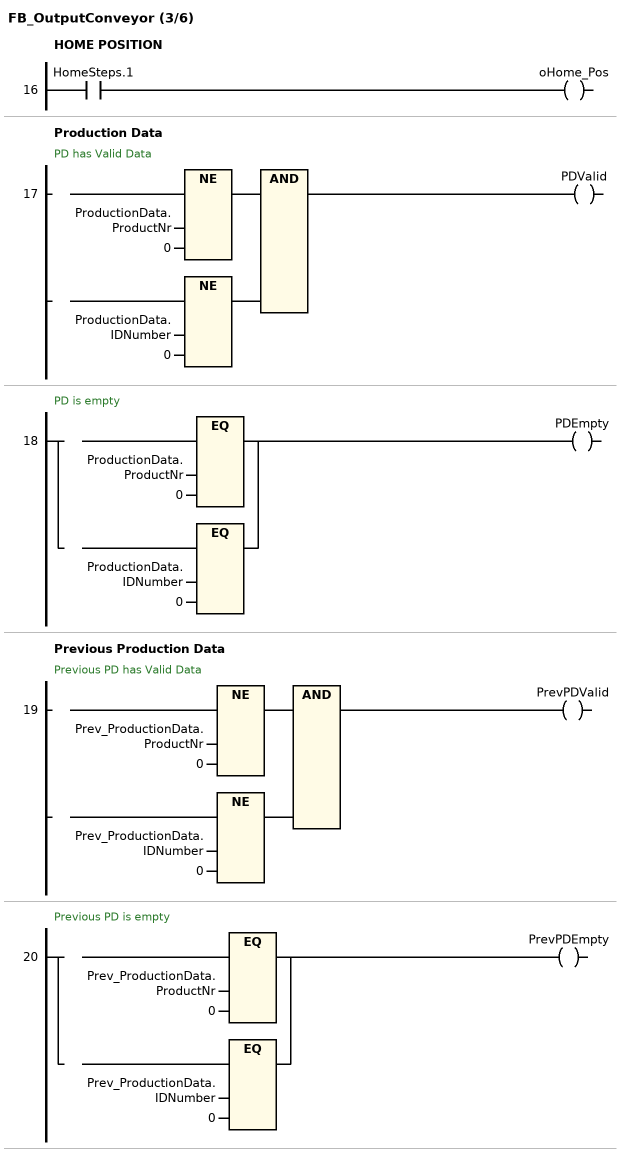
// NETWORK 16: HOME POSITION
oHome_Pos := HomeSteps.1;

// NETWORK 17: Production Data
// PD has Valid Data
PDValid := ProductionData.ProductNr <> 0 AND ProductionData.IDNumber <> 0;

// NETWORK 18
// PD is empty
PDEmpty := ProductionData.ProductNr = 0 OR ProductionData.IDNumber = 0;

// NETWORK 19: Previous Production Data
// Previous PD has Valid Data
PrevPDValid := Prev_ProductionData.ProductNr <> 0 AND Prev_ProductionData.IDNumber <> 0;

// NETWORK 20
// Previous PD is empty
PrevPDEmpty := Prev_ProductionData.ProductNr = 0 OR Prev_ProductionData.IDNumber = 0;

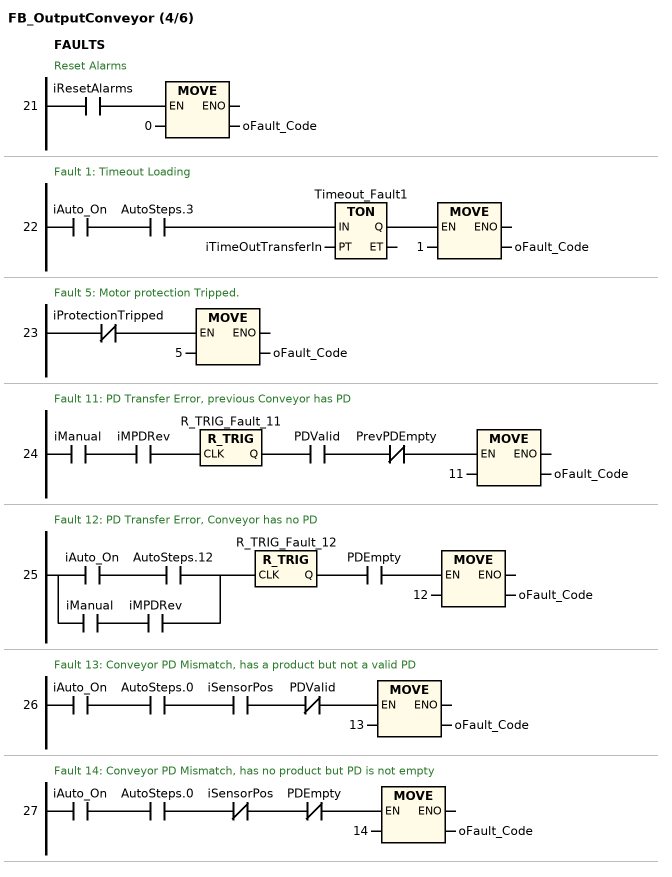
// NETWORK 21: FAULTS
// Reset Alarms
IF iResetAlarms THEN oFault_Code := 0; END_IF

// NETWORK 22
// Fault 1: Timeout Loading
Timeout_Fault1(IN := iAuto_On AND AutoSteps.3, PT := iTimeOutTransferIn); // TON
IF Timeout_Fault1.Q THEN oFault_Code := 1; END_IF

// NETWORK 23
// Fault 5: Motor protection Tripped.
IF NOT iProtectionTripped THEN oFault_Code := 5; END_IF

// NETWORK 24
// Fault 11: PD Transfer Error, previous Conveyor has PD
R_TRIG_Fault_11(CLK := iManual AND iMPDRev); // R_TRIG
IF R_TRIG_Fault_11.Q AND PDValid AND NOT PrevPDEmpty THEN oFault_Code := 11; END_IF

// NETWORK 25
// Fault 12: PD Transfer Error, Conveyor has no PD
R_TRIG_Fault_12(CLK := iAuto_On AND AutoSteps.12 OR iManual AND iMPDRev); // R_TRIG
IF R_TRIG_Fault_12.Q AND PDEmpty THEN oFault_Code := 12; END_IF

// NETWORK 26
// Fault 13: Conveyor PD Mismatch, has a product but not a valid PD
IF iAuto_On AND AutoSteps.0 AND iSensorPos AND NOT PDValid THEN oFault_Code := 13; END_IF

// NETWORK 27
// Fault 14: Conveyor PD Mismatch, has no product but PD is not empty
IF iAuto_On AND AutoSteps.0 AND NOT iSensorPos AND NOT PDEmpty THEN oFault_Code := 14; END_IF

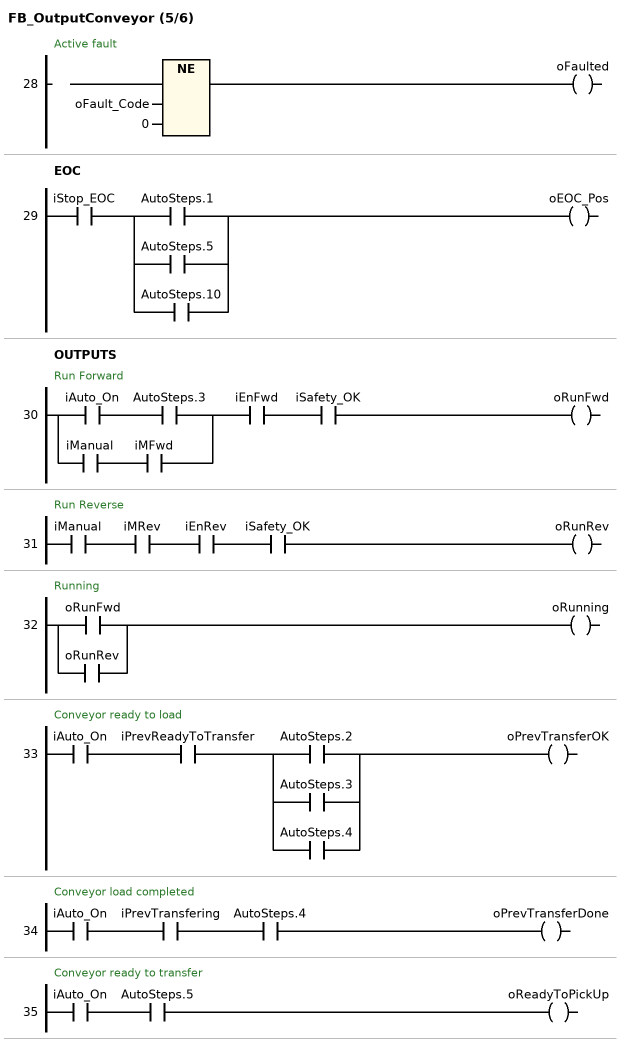
// NETWORK 28
// Active fault
oFaulted := oFault_Code <> 0;

// NETWORK 29: EOC
oEOC_Pos := iStop_EOC AND (AutoSteps.1 OR AutoSteps.5 OR AutoSteps.10);

// NETWORK 30: OUTPUTS
// Run Forward
oRunFwd := (iAuto_On AND AutoSteps.3 OR iManual AND iMFwd) AND iEnFwd AND iSafety_OK;

// NETWORK 31
// Run Reverse
oRunRev := iManual AND iMRev AND iEnRev AND iSafety_OK;

// NETWORK 32
// Running
oRunning := oRunFwd OR oRunRev;

// NETWORK 33
// Conveyor ready to load
oPrevTransferOK := iAuto_On AND iPrevReadyToTransfer AND (AutoSteps.2 OR AutoSteps.3 OR AutoSteps.4);

// NETWORK 34
// Conveyor load completed
oPrevTransferDone := iAuto_On AND iPrevTransfering AND AutoSteps.4;

// NETWORK 35
// Conveyor ready to transfer
oReadyToPickUp := iAuto_On AND AutoSteps.5;

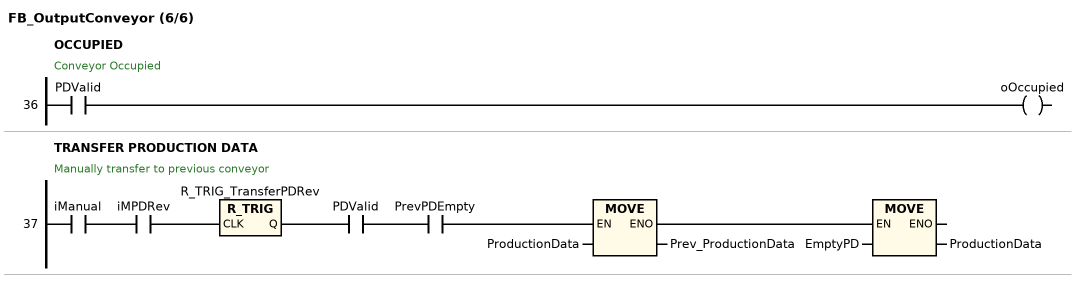
// NETWORK 36: OCCUPIED
// Conveyor Occupied
oOccupied := PDValid;

// NETWORK 37: TRANSFER PRODUCTION DATA
// Manually transfer to previous conveyor
R_TRIG_TransferPDRev(CLK := iManual AND iMPDRev); // R_TRIG
_w13 := R_TRIG_TransferPDRev.Q AND PDValid AND PrevPDEmpty;
IF _w13 THEN Prev_ProductionData := ProductionData; END_IF
IF _w13 THEN ProductionData := EmptyPD; END_IF

END_FUNCTION_BLOCK

// Device/Application/SOP670
PROGRAM SOP670
VAR
END_VAR

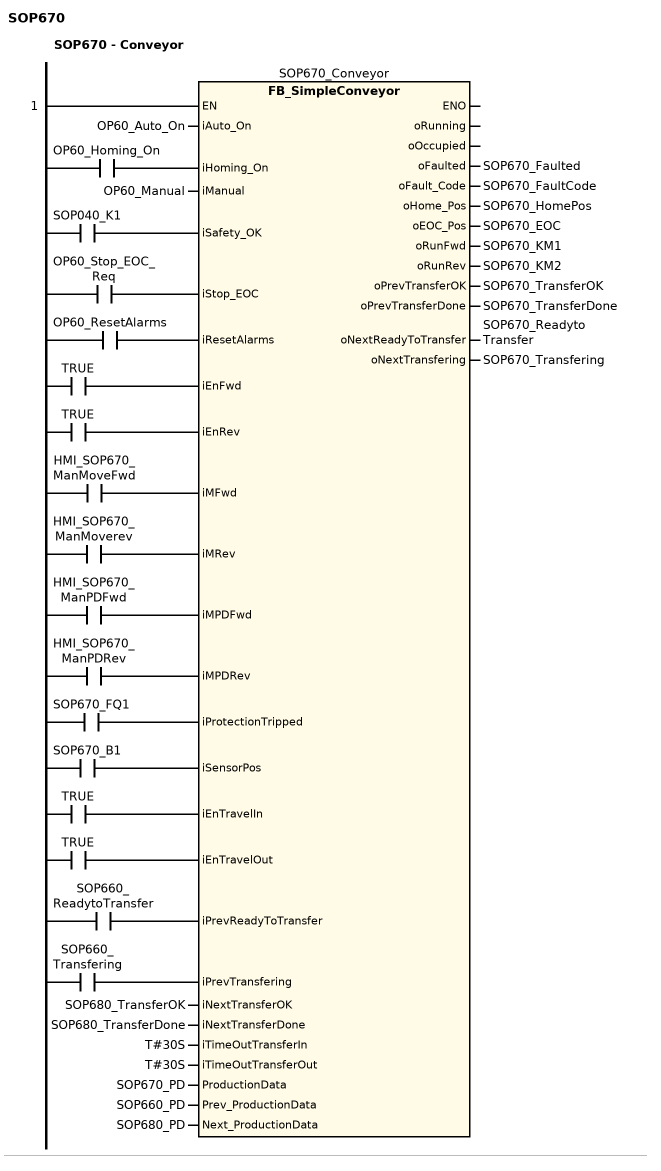
// NETWORK 1: SOP670 - Conveyor
SOP670_Conveyor(
    iAuto_On := OP60_Auto_On,
    iHoming_On := OP60_Homing_On,
    iManual := OP60_Manual,
    iSafety_OK := SOP040_K1,
    iStop_EOC := OP60_Stop_EOC_Req,
    iResetAlarms := OP60_ResetAlarms,
    iEnFwd := TRUE,
    iEnRev := TRUE,
    iMFwd := HMI_SOP670_ManMoveFwd,
    iMRev := HMI_SOP670_ManMoverev,
    iMPDFwd := HMI_SOP670_ManPDFwd,
    iMPDRev := HMI_SOP670_ManPDRev,
    iProtectionTripped := SOP670_FQ1,
    iSensorPos := SOP670_B1,
    iEnTravelIn := TRUE,
    iEnTravelOut := TRUE,
    iPrevReadyToTransfer := SOP660_ReadytoTransfer,
    iPrevTransfering := SOP660_Transfering,
    iNextTransferOK := SOP680_TransferOK,
    iNextTransferDone := SOP680_TransferDone,
    iTimeOutTransferIn := T#30S,
    iTimeOutTransferOut := T#30S,
    ProductionData := SOP670_PD,
    Prev_ProductionData := SOP660_PD,
    Next_ProductionData := SOP680_PD,
    oFaulted => SOP670_Faulted,
    oFault_Code => SOP670_FaultCode,
    oHome_Pos => SOP670_HomePos,
    oEOC_Pos => SOP670_EOC,
    oRunFwd => SOP670_KM1,
    oRunRev => SOP670_KM2,
    oPrevTransferOK => SOP670_TransferOK,
    oPrevTransferDone => SOP670_TransferDone,
    oNextReadyToTransfer => SOP670_ReadytoTransfer,
    oNextTransfering => SOP670_Transfering); // FB_SimpleConveyor

END_PROGRAM

// Device/Application/FBs/FB_SimpleConveyor
FUNCTION_BLOCK FB_SimpleConveyor
VAR_INPUT
	iAuto_On: BOOL; // Auto-On cycle active
	iHoming_On: BOOL; // Homing-On cycle active
	iManual: BOOL; // Manual mode active
	iSafety_OK: BOOL; // Safety circuit OK
	iStop_EOC: BOOL; // Stop EOC selected
	iResetAlarms: BOOL; // Reset Alarms
	
	iEnFwd: BOOL := TRUE; // Interlock signal movement forward
	iEnRev: BOOL := TRUE; // Interlock signal movement reverse
	
	iMFwd: BOOL; 	// Manual Fwd request
	iMRev: BOOL; 	// Manual Rev request
	iMPDFwd: BOOL; 	// Manual Move PD forward
	iMPDRev: BOOL; 	// Manual Move PD reverse
	
	iProtectionTripped: BOOL := FALSE; // Motor Protection Tripped
	
	iSensorPos: BOOL; // Product in position
	
	iEnTravelIn: BOOL := TRUE; // Enable product transfer from previous conveyor.
	iEnTravelOut: BOOL := TRUE; // Enable product transfer to next conveyor.
	
	iPrevReadyToTransfer: BOOL; // Previous conveyor ready to transfer
	iPrevTransfering: BOOL; // Previous conveyor transfering
	iNextTransferOK: BOOL; // Next conveyor ready to load
	iNextTransferDone: BOOL;  // Next conveyor transfer done
	
	iTimeOutTransferIn: TIME := T#10S; // Time out time for transfer in
	iTimeOutTransferOut: TIME := T#10S; // Time out time for transfer out
END_VAR
VAR_IN_OUT
	ProductionData: ProductionData; 		// Production Data
	Prev_ProductionData: ProductionData;	// Previous Production Data
	Next_ProductionData: ProductionData;	// Next Production Data
END_VAR
VAR_OUTPUT
	oRunning: BOOL; // Conveyor Running
	oOccupied: BOOL; // Conveyor Occupied
	oFaulted : BOOL; // Conveyor faulted
	oFault_Code: INT; // Conveyor fault code
	oHome_Pos: BOOL; // Conveyor Home Position reached
	oEOC_Pos: BOOL; // Conveyor Stop EOC reached

	oRunFwd: BOOL; // Conveyor running forward
	oRunRev: BOOL; // Conveyor running reverse	

	oPrevTransferOK: BOOL; // Conveyor ready to load
	oPrevTransferDone: BOOL; // Conveyor load completed
	oNextReadyToTransfer: BOOL; // Conveyor ready to transfer
	oNextTransfering: BOOL; // Conveyor transfering
END_VAR
VAR
	AutoSteps: WORD;
	HomeSteps: WORD;
	
	Timeout_Fault1: TON;
	Timeout_Fault2: TON;
	
	EmptyPD: ProductionData;
	PDValid: BOOL;		// PD is Valid
	PDEmpty: BOOL;		// PD is Empty
	PrevPDValid: BOOL;	// Previous PD is Valid
	PrevPDEmpty: BOOL;	// Previous PD is Empty
	NextPDValid: BOOL;	// Next PD is Valid
	NextPDEmpty: BOOL;	// Next PD is Empty
	R_TRIG_TransferPDFwd: R_TRIG;
	R_TRIG_TransferPDRev: R_TRIG;
	R_TRIG_Fault_10: R_TRIG;
	R_TRIG_Fault_11: R_TRIG;
	R_TRIG_Fault_12: R_TRIG;
END_VAR
VAR // added by the converter: edge detectors and wires of the graphical bodies
    _w1, _w2, _w3, _w4, _w5, _w6, _w7, _w8, _w9, _w10, _w11, _w12, _w13, _w14, _w15, _w16 : BOOL;
END_VAR

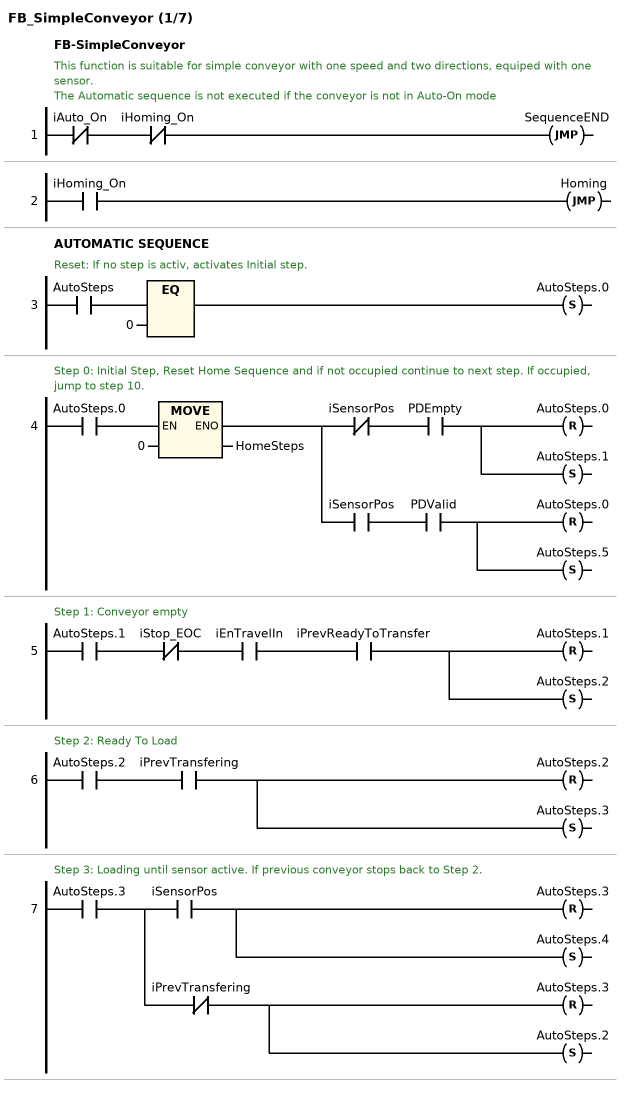
// NETWORK 1: FB-SimpleConveyor
// This function is suitable for simple conveyor with one speed and two directions, equiped with one sensor.
//
// The Automatic sequence is not executed if the conveyor is not in Auto-On mode
IF NOT iAuto_On AND NOT iHoming_On THEN JMP SequenceEND; END_IF

// NETWORK 2
IF iHoming_On THEN JMP Homing; END_IF

// NETWORK 3: AUTOMATIC SEQUENCE
// Reset: If no step is activ, activates Initial step.
AutoSteps.0 S= AutoSteps = 0;

// NETWORK 4
// Step 0: Initial Step, Reset Home Sequence and if not occupied continue to next step. If occupied, jump to step 10.
_w1 := AutoSteps.0;
IF _w1 THEN HomeSteps := 0; END_IF
_w2 := _w1 AND NOT iSensorPos AND PDEmpty;
AutoSteps.0 R= _w2;
AutoSteps.1 S= _w2;
_w3 := _w1 AND iSensorPos AND PDValid;
AutoSteps.0 R= _w3;
AutoSteps.5 S= _w3;

// NETWORK 5
// Step 1: Conveyor empty
_w4 := AutoSteps.1 AND NOT iStop_EOC AND iEnTravelIn AND iPrevReadyToTransfer;
AutoSteps.1 R= _w4;
AutoSteps.2 S= _w4;

// NETWORK 6
// Step 2: Ready To Load
_w5 := AutoSteps.2 AND iPrevTransfering;
AutoSteps.2 R= _w5;
AutoSteps.3 S= _w5;

// NETWORK 7
// Step 3: Loading until sensor active. If previous conveyor stops back to Step 2.
_w6 := AutoSteps.3;
_w7 := _w6 AND iSensorPos;
AutoSteps.3 R= _w7;
AutoSteps.4 S= _w7;
_w8 := _w6 AND NOT iPrevTransfering;
AutoSteps.3 R= _w8;
AutoSteps.2 S= _w8;

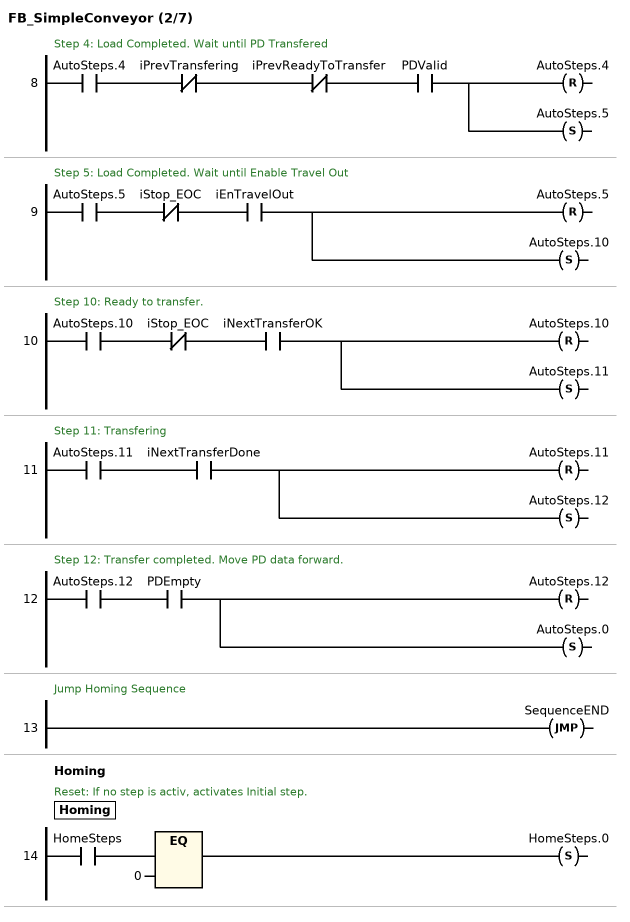
// NETWORK 8
// Step 4: Load Completed. Wait until PD Transfered
_w9 := AutoSteps.4 AND NOT iPrevTransfering AND NOT iPrevReadyToTransfer AND PDValid;
AutoSteps.4 R= _w9;
AutoSteps.5 S= _w9;

// NETWORK 9
// Step 5: Load Completed. Wait until Enable Travel Out
_w10 := AutoSteps.5 AND NOT iStop_EOC AND iEnTravelOut;
AutoSteps.5 R= _w10;
AutoSteps.10 S= _w10;

// NETWORK 10
// Step 10: Ready to transfer.
_w11 := AutoSteps.10 AND NOT iStop_EOC AND iNextTransferOK;
AutoSteps.10 R= _w11;
AutoSteps.11 S= _w11;

// NETWORK 11
// Step 11: Transfering
_w12 := AutoSteps.11 AND iNextTransferDone;
AutoSteps.11 R= _w12;
AutoSteps.12 S= _w12;

// NETWORK 12
// Step 12: Transfer completed. Move PD data forward.
_w13 := AutoSteps.12 AND PDEmpty;
AutoSteps.12 R= _w13;
AutoSteps.0 S= _w13;

// NETWORK 13
// Jump Homing Sequence
JMP SequenceEND;

// NETWORK 14: Homing
// Reset: If no step is activ, activates Initial step.
Homing:
HomeSteps.0 S= HomeSteps = 0;

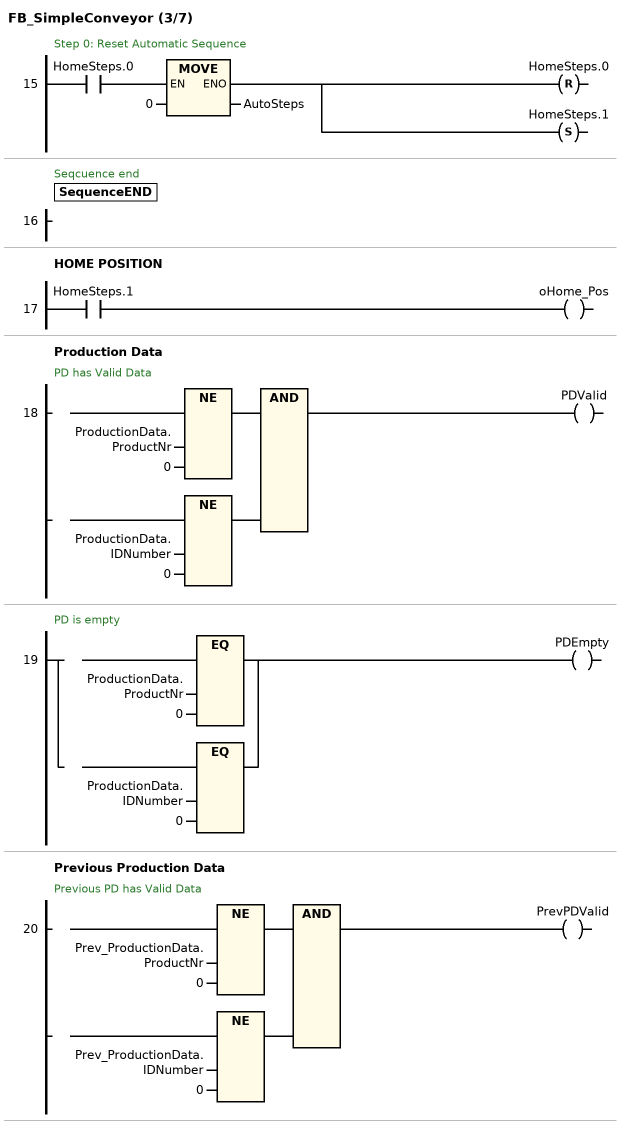
// NETWORK 15
// Step 0: Reset Automatic Sequence
_w14 := HomeSteps.0;
IF _w14 THEN AutoSteps := 0; END_IF
HomeSteps.0 R= _w14;
HomeSteps.1 S= _w14;

// NETWORK 16
// Seqcuence end
SequenceEND: ;

// NETWORK 17: HOME POSITION
oHome_Pos := HomeSteps.1;

// NETWORK 18: Production Data
// PD has Valid Data
PDValid := ProductionData.ProductNr <> 0 AND ProductionData.IDNumber <> 0;

// NETWORK 19
// PD is empty
PDEmpty := ProductionData.ProductNr = 0 OR ProductionData.IDNumber = 0;

// NETWORK 20: Previous Production Data
// Previous PD has Valid Data
PrevPDValid := Prev_ProductionData.ProductNr <> 0 AND Prev_ProductionData.IDNumber <> 0;

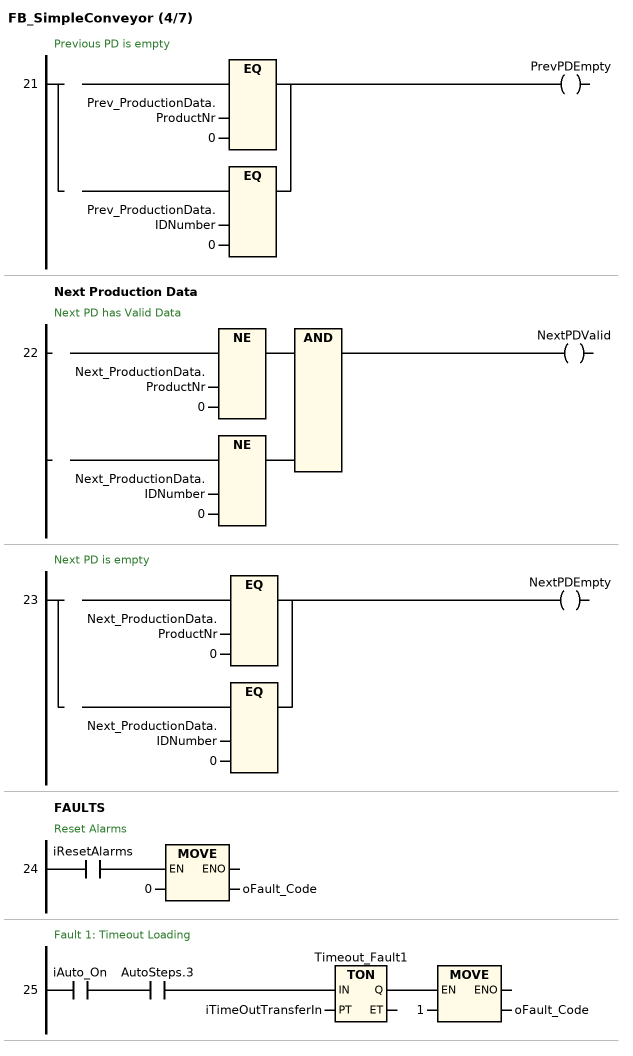
// NETWORK 21
// Previous PD is empty
PrevPDEmpty := Prev_ProductionData.ProductNr = 0 OR Prev_ProductionData.IDNumber = 0;

// NETWORK 22: Next Production Data
// Next PD has Valid Data
NextPDValid := Next_ProductionData.ProductNr <> 0 AND Next_ProductionData.IDNumber <> 0;

// NETWORK 23
// Next PD is empty
NextPDEmpty := Next_ProductionData.ProductNr = 0 OR Next_ProductionData.IDNumber = 0;

// NETWORK 24: FAULTS
// Reset Alarms
IF iResetAlarms THEN oFault_Code := 0; END_IF

// NETWORK 25
// Fault 1: Timeout Loading
Timeout_Fault1(IN := iAuto_On AND AutoSteps.3, PT := iTimeOutTransferIn); // TON
IF Timeout_Fault1.Q THEN oFault_Code := 1; END_IF

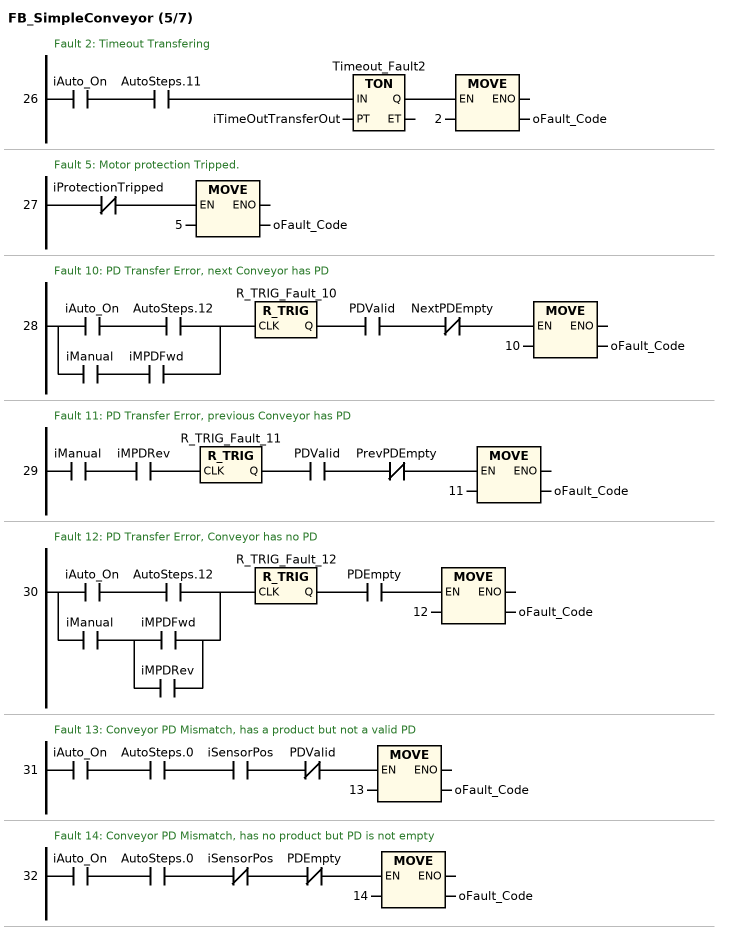
// NETWORK 26
// Fault 2: Timeout Transfering
Timeout_Fault2(IN := iAuto_On AND AutoSteps.11, PT := iTimeOutTransferOut); // TON
IF Timeout_Fault2.Q THEN oFault_Code := 2; END_IF

// NETWORK 27
// Fault 5: Motor protection Tripped.
IF NOT iProtectionTripped THEN oFault_Code := 5; END_IF

// NETWORK 28
// Fault 10: PD Transfer Error, next Conveyor has PD
R_TRIG_Fault_10(CLK := iAuto_On AND AutoSteps.12 OR iManual AND iMPDFwd); // R_TRIG
IF R_TRIG_Fault_10.Q AND PDValid AND NOT NextPDEmpty THEN oFault_Code := 10; END_IF

// NETWORK 29
// Fault 11: PD Transfer Error, previous Conveyor has PD
R_TRIG_Fault_11(CLK := iManual AND iMPDRev); // R_TRIG
IF R_TRIG_Fault_11.Q AND PDValid AND NOT PrevPDEmpty THEN oFault_Code := 11; END_IF

// NETWORK 30
// Fault 12: PD Transfer Error, Conveyor has no PD
R_TRIG_Fault_12(CLK := iAuto_On AND AutoSteps.12 OR iManual AND (iMPDFwd OR iMPDRev)); // R_TRIG
IF R_TRIG_Fault_12.Q AND PDEmpty THEN oFault_Code := 12; END_IF

// NETWORK 31
// Fault 13: Conveyor PD Mismatch, has a product but not a valid PD
IF iAuto_On AND AutoSteps.0 AND iSensorPos AND NOT PDValid THEN oFault_Code := 13; END_IF

// NETWORK 32
// Fault 14: Conveyor PD Mismatch, has no product but PD is not empty
IF iAuto_On AND AutoSteps.0 AND NOT iSensorPos AND NOT PDEmpty THEN oFault_Code := 14; END_IF

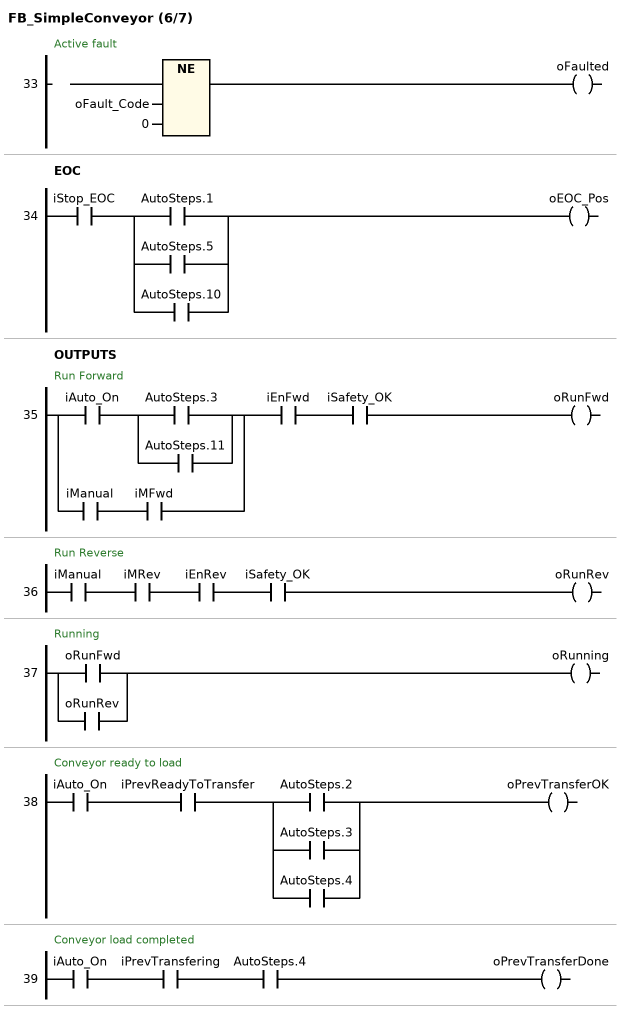
// NETWORK 33
// Active fault
oFaulted := oFault_Code <> 0;

// NETWORK 34: EOC
oEOC_Pos := iStop_EOC AND (AutoSteps.1 OR AutoSteps.5 OR AutoSteps.10);

// NETWORK 35: OUTPUTS
// Run Forward
oRunFwd := (iAuto_On AND (AutoSteps.3 OR AutoSteps.11) OR iManual AND iMFwd) AND iEnFwd AND iSafety_OK;

// NETWORK 36
// Run Reverse
oRunRev := iManual AND iMRev AND iEnRev AND iSafety_OK;

// NETWORK 37
// Running
oRunning := oRunFwd OR oRunRev;

// NETWORK 38
// Conveyor ready to load
oPrevTransferOK := iAuto_On AND iPrevReadyToTransfer AND (AutoSteps.2 OR AutoSteps.3 OR AutoSteps.4);

// NETWORK 39
// Conveyor load completed
oPrevTransferDone := iAuto_On AND iPrevTransfering AND AutoSteps.4;

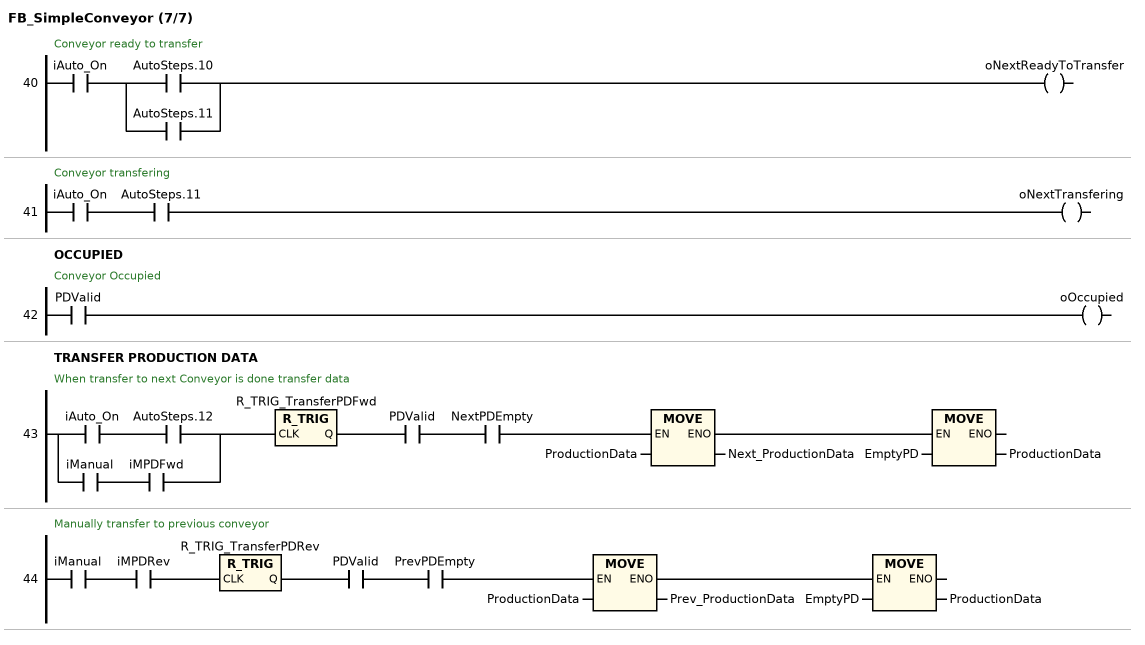
// NETWORK 40
// Conveyor ready to transfer
oNextReadyToTransfer := iAuto_On AND (AutoSteps.10 OR AutoSteps.11);

// NETWORK 41
// Conveyor transfering
oNextTransfering := iAuto_On AND AutoSteps.11;

// NETWORK 42: OCCUPIED
// Conveyor Occupied
oOccupied := PDValid;

// NETWORK 43: TRANSFER PRODUCTION DATA
// When transfer to next Conveyor is done transfer data
R_TRIG_TransferPDFwd(CLK := iAuto_On AND AutoSteps.12 OR iManual AND iMPDFwd); // R_TRIG
_w15 := R_TRIG_TransferPDFwd.Q AND PDValid AND NextPDEmpty;
IF _w15 THEN Next_ProductionData := ProductionData; END_IF
IF _w15 THEN ProductionData := EmptyPD; END_IF

// NETWORK 44
// Manually transfer to previous conveyor
R_TRIG_TransferPDRev(CLK := iManual AND iMPDRev); // R_TRIG
_w16 := R_TRIG_TransferPDRev.Q AND PDValid AND PrevPDEmpty;
IF _w16 THEN Prev_ProductionData := ProductionData; END_IF
IF _w16 THEN ProductionData := EmptyPD; END_IF

END_FUNCTION_BLOCK

// Device/Application/SOP660
PROGRAM SOP660
VAR
END_VAR

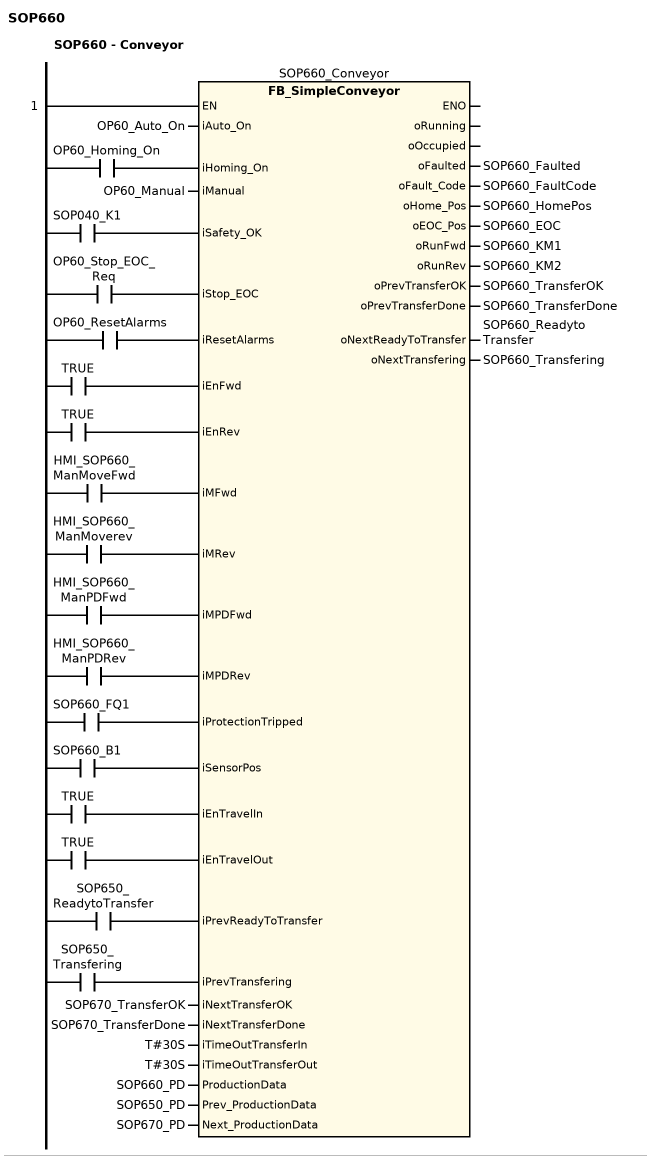
// NETWORK 1: SOP660 - Conveyor
SOP660_Conveyor(
    iAuto_On := OP60_Auto_On,
    iHoming_On := OP60_Homing_On,
    iManual := OP60_Manual,
    iSafety_OK := SOP040_K1,
    iStop_EOC := OP60_Stop_EOC_Req,
    iResetAlarms := OP60_ResetAlarms,
    iEnFwd := TRUE,
    iEnRev := TRUE,
    iMFwd := HMI_SOP660_ManMoveFwd,
    iMRev := HMI_SOP660_ManMoverev,
    iMPDFwd := HMI_SOP660_ManPDFwd,
    iMPDRev := HMI_SOP660_ManPDRev,
    iProtectionTripped := SOP660_FQ1,
    iSensorPos := SOP660_B1,
    iEnTravelIn := TRUE,
    iEnTravelOut := TRUE,
    iPrevReadyToTransfer := SOP650_ReadytoTransfer,
    iPrevTransfering := SOP650_Transfering,
    iNextTransferOK := SOP670_TransferOK,
    iNextTransferDone := SOP670_TransferDone,
    iTimeOutTransferIn := T#30S,
    iTimeOutTransferOut := T#30S,
    ProductionData := SOP660_PD,
    Prev_ProductionData := SOP650_PD,
    Next_ProductionData := SOP670_PD,
    oFaulted => SOP660_Faulted,
    oFault_Code => SOP660_FaultCode,
    oHome_Pos => SOP660_HomePos,
    oEOC_Pos => SOP660_EOC,
    oRunFwd => SOP660_KM1,
    oRunRev => SOP660_KM2,
    oPrevTransferOK => SOP660_TransferOK,
    oPrevTransferDone => SOP660_TransferDone,
    oNextReadyToTransfer => SOP660_ReadytoTransfer,
    oNextTransfering => SOP660_Transfering); // FB_SimpleConveyor

END_PROGRAM

// Device/Application/SOP650
PROGRAM SOP650
VAR
END_VAR

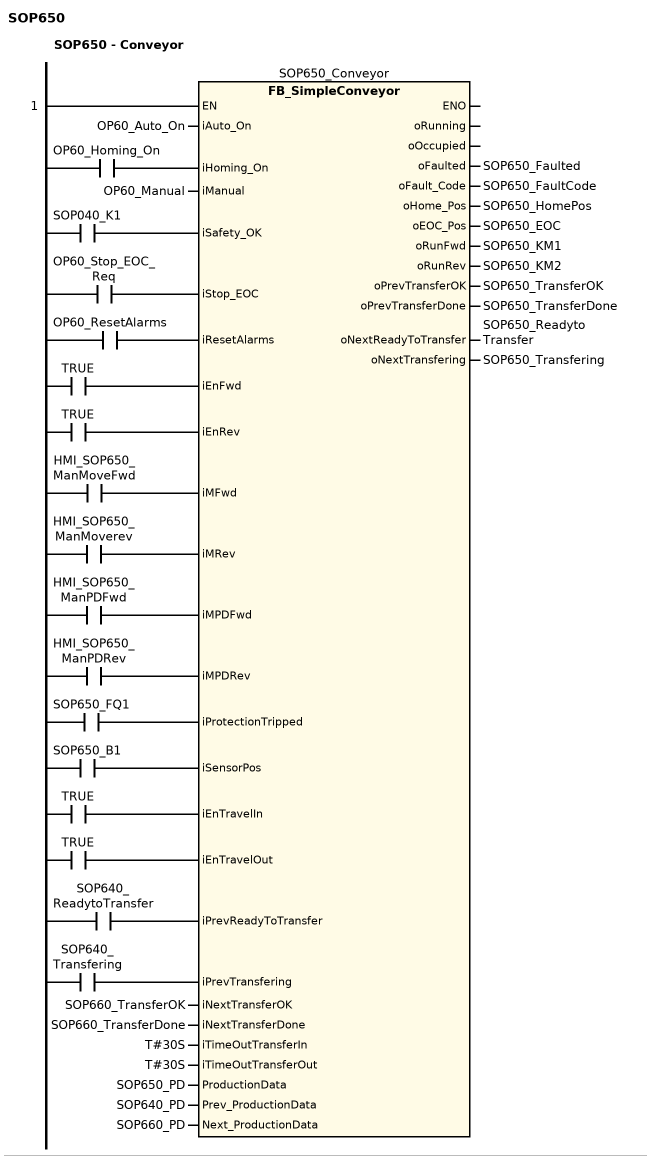
// NETWORK 1: SOP650 - Conveyor
SOP650_Conveyor(
    iAuto_On := OP60_Auto_On,
    iHoming_On := OP60_Homing_On,
    iManual := OP60_Manual,
    iSafety_OK := SOP040_K1,
    iStop_EOC := OP60_Stop_EOC_Req,
    iResetAlarms := OP60_ResetAlarms,
    iEnFwd := TRUE,
    iEnRev := TRUE,
    iMFwd := HMI_SOP650_ManMoveFwd,
    iMRev := HMI_SOP650_ManMoverev,
    iMPDFwd := HMI_SOP650_ManPDFwd,
    iMPDRev := HMI_SOP650_ManPDRev,
    iProtectionTripped := SOP650_FQ1,
    iSensorPos := SOP650_B1,
    iEnTravelIn := TRUE,
    iEnTravelOut := TRUE,
    iPrevReadyToTransfer := SOP640_ReadytoTransfer,
    iPrevTransfering := SOP640_Transfering,
    iNextTransferOK := SOP660_TransferOK,
    iNextTransferDone := SOP660_TransferDone,
    iTimeOutTransferIn := T#30S,
    iTimeOutTransferOut := T#30S,
    ProductionData := SOP650_PD,
    Prev_ProductionData := SOP640_PD,
    Next_ProductionData := SOP660_PD,
    oFaulted => SOP650_Faulted,
    oFault_Code => SOP650_FaultCode,
    oHome_Pos => SOP650_HomePos,
    oEOC_Pos => SOP650_EOC,
    oRunFwd => SOP650_KM1,
    oRunRev => SOP650_KM2,
    oPrevTransferOK => SOP650_TransferOK,
    oPrevTransferDone => SOP650_TransferDone,
    oNextReadyToTransfer => SOP650_ReadytoTransfer,
    oNextTransfering => SOP650_Transfering); // FB_SimpleConveyor

END_PROGRAM

// Device/Application/SOP640
PROGRAM SOP640
VAR
	OP60_CYCLE_TIME: TON;
	TON_0: TON;
	TimerON_0: TIME;
	
	SOP640_Occupied: BOOL;
	SOP640_BoxWaiting: BOOL;
	OP60_LastCycleTime_Str: STRING;
	RS_0: RS;
	SR_publish: BOOL;
	R_TRIG_0: R_TRIG;
	
	MB16: BOOL;
	MB16T: BOOL;
	MB20: BOOL;
	MB24: BOOL;
	
	Product_str: STRING(1024);
	R_TRIG_1: R_TRIG;
	R_TRIG_2: R_TRIG;
	R_TRIG_3: R_TRIG;
	R_TRIG_4: R_TRIG;
	RS_1: RS;
	R_TRIG_5: R_TRIG;
	R_TRIG_6: R_TRIG;
	R_TRIG_7: R_TRIG;
	R_TRIG_8: R_TRIG;
END_VAR
VAR // added by the converter: edge detectors and wires of the graphical bodies
    _w1, _w2, _w3, _w4, _w5, _w6, _w7, _w8, _w9, _w10 : BOOL;
    _ft1 : F_TRIG;
    _rt1 : R_TRIG;
END_VAR

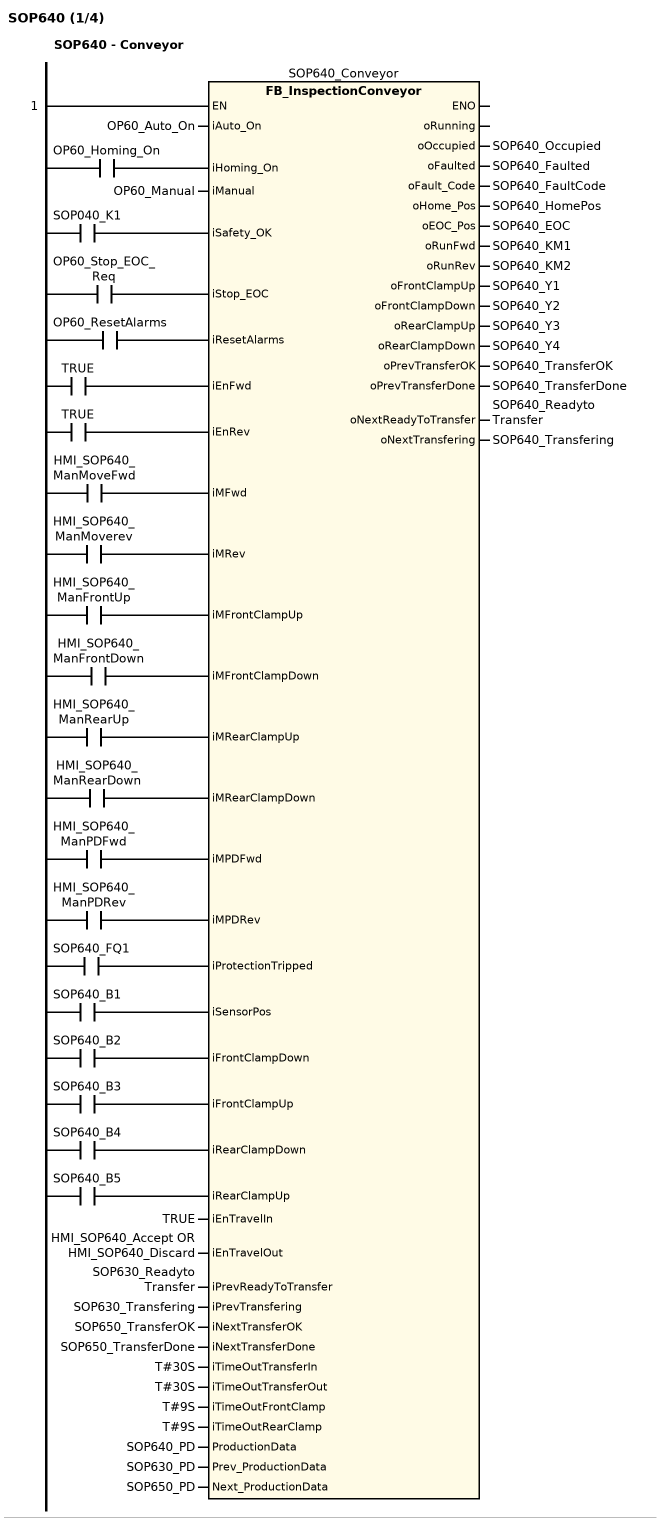
// NETWORK 1: SOP640 - Conveyor
SOP640_Conveyor(
    iAuto_On := OP60_Auto_On,
    iHoming_On := OP60_Homing_On,
    iManual := OP60_Manual,
    iSafety_OK := SOP040_K1,
    iStop_EOC := OP60_Stop_EOC_Req,
    iResetAlarms := OP60_ResetAlarms,
    iEnFwd := TRUE,
    iEnRev := TRUE,
    iMFwd := HMI_SOP640_ManMoveFwd,
    iMRev := HMI_SOP640_ManMoverev,
    iMFrontClampUp := HMI_SOP640_ManFrontUp,
    iMFrontClampDown := HMI_SOP640_ManFrontDown,
    iMRearClampUp := HMI_SOP640_ManRearUp,
    iMRearClampDown := HMI_SOP640_ManRearDown,
    iMPDFwd := HMI_SOP640_ManPDFwd,
    iMPDRev := HMI_SOP640_ManPDRev,
    iProtectionTripped := SOP640_FQ1,
    iSensorPos := SOP640_B1,
    iFrontClampDown := SOP640_B2,
    iFrontClampUp := SOP640_B3,
    iRearClampDown := SOP640_B4,
    iRearClampUp := SOP640_B5,
    iEnTravelIn := TRUE,
    iEnTravelOut := HMI_SOP640_Accept OR HMI_SOP640_Discard,
    iPrevReadyToTransfer := SOP630_ReadytoTransfer,
    iPrevTransfering := SOP630_Transfering,
    iNextTransferOK := SOP650_TransferOK,
    iNextTransferDone := SOP650_TransferDone,
    iTimeOutTransferIn := T#30S,
    iTimeOutTransferOut := T#30S,
    iTimeOutFrontClamp := T#9S,
    iTimeOutRearClamp := T#9S,
    ProductionData := SOP640_PD,
    Prev_ProductionData := SOP630_PD,
    Next_ProductionData := SOP650_PD,
    oOccupied => SOP640_Occupied,
    oFaulted => SOP640_Faulted,
    oFault_Code => SOP640_FaultCode,
    oHome_Pos => SOP640_HomePos,
    oEOC_Pos => SOP640_EOC,
    oRunFwd => SOP640_KM1,
    oRunRev => SOP640_KM2,
    oFrontClampUp => SOP640_Y1,
    oFrontClampDown => SOP640_Y2,
    oRearClampUp => SOP640_Y3,
    oRearClampDown => SOP640_Y4,
    oPrevTransferOK => SOP640_TransferOK,
    oPrevTransferDone => SOP640_TransferDone,
    oNextReadyToTransfer => SOP640_ReadytoTransfer,
    oNextTransfering => SOP640_Transfering); // FB_InspectionConveyor

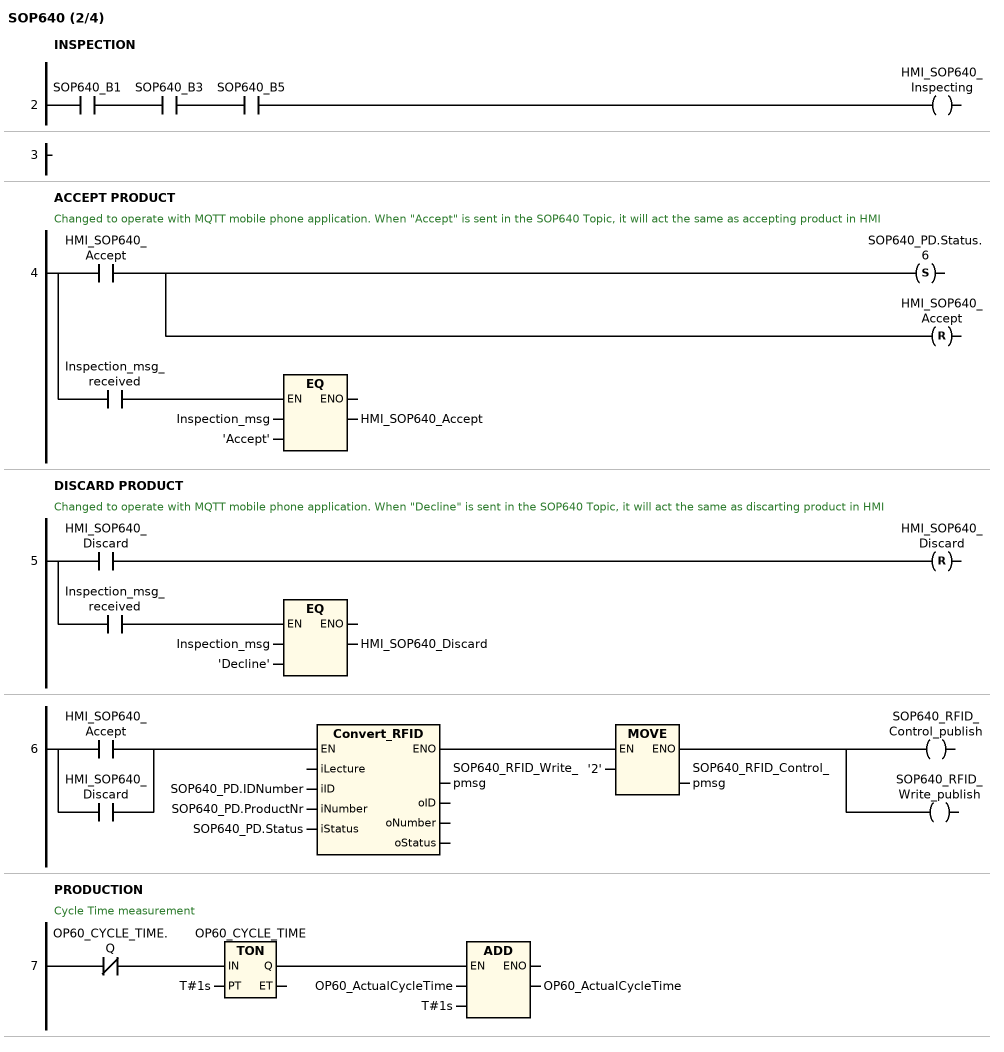
// NETWORK 2: INSPECTION
HMI_SOP640_Inspecting := SOP640_B1 AND SOP640_B3 AND SOP640_B5;

// NETWORK 3

// NETWORK 4: ACCEPT PRODUCT
// Changed to operate with MQTT mobile phone application. When "Accept" is sent in the SOP640 Topic, it will act the same as accepting product in HMI
_w1 := HMI_SOP640_Accept;
SOP640_PD.Status.6 S= _w1;
HMI_SOP640_Accept R= _w1;
IF Inspection_msg_received THEN HMI_SOP640_Accept := Inspection_msg = 'Accept'; END_IF

// NETWORK 5: DISCARD PRODUCT
// Changed to operate with MQTT mobile phone application. When "Decline" is sent in the SOP640 Topic, it will act the same as discarting product in HMI
HMI_SOP640_Discard R= HMI_SOP640_Discard;
IF Inspection_msg_received THEN HMI_SOP640_Discard := Inspection_msg = 'Decline'; END_IF

// NETWORK 6
_w2 := HMI_SOP640_Accept OR HMI_SOP640_Discard;
IF _w2 THEN
    SOP640_RFID_Write_pmsg := Convert_RFID(iID := SOP640_PD.IDNumber, iNumber := SOP640_PD.ProductNr, iStatus := SOP640_PD.Status);
END_IF
IF _w2 THEN SOP640_RFID_Control_pmsg := '2'; END_IF
SOP640_RFID_Control_publish := _w2;
SOP640_RFID_Write_publish := _w2;

// NETWORK 7: PRODUCTION
// Cycle Time measurement
OP60_CYCLE_TIME(IN := NOT OP60_CYCLE_TIME.Q, PT := T#1s); // TON
IF OP60_CYCLE_TIME.Q THEN OP60_ActualCycleTime := OP60_ActualCycleTime + T#1s; END_IF

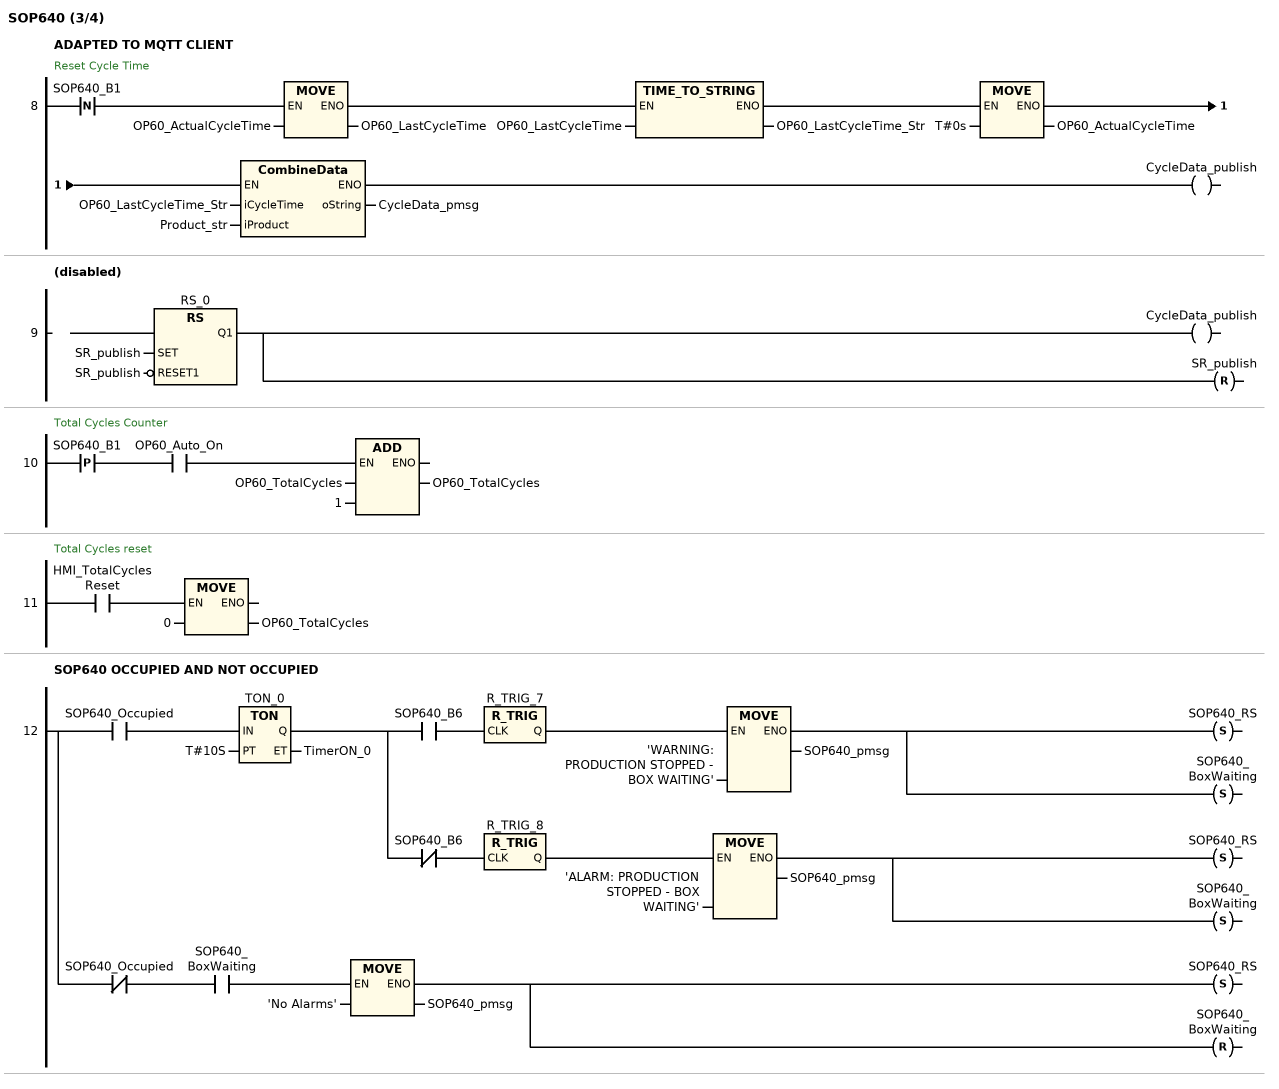
// NETWORK 8: ADAPTED TO MQTT CLIENT
// Reset Cycle Time
_ft1(CLK := SOP640_B1);
_w3 := _ft1.Q;
IF _w3 THEN OP60_LastCycleTime := OP60_ActualCycleTime; END_IF
IF _w3 THEN OP60_LastCycleTime_Str := TIME_TO_STRING(OP60_LastCycleTime); END_IF
IF _w3 THEN OP60_ActualCycleTime := T#0s; END_IF
IF _w3 THEN
    CombineData(iCycleTime := OP60_LastCycleTime_Str, iProduct := Product_str, oString => CycleData_pmsg);
END_IF
CycleData_publish := _w3;

// NETWORK 9 (disabled)
// RS_0(SET := SR_publish, RESET1 := NOT SR_publish); // RS
// CycleData_publish := RS_0.Q1;
// SR_publish R= RS_0.Q1;

// NETWORK 10
// Total Cycles Counter
_rt1(CLK := SOP640_B1);
IF _rt1.Q AND OP60_Auto_On THEN OP60_TotalCycles := OP60_TotalCycles + 1; END_IF

// NETWORK 11
// Total Cycles reset
IF HMI_TotalCyclesReset THEN OP60_TotalCycles := 0; END_IF

// NETWORK 12: SOP640 OCCUPIED AND NOT OCCUPIED
TON_0(IN := SOP640_Occupied, PT := T#10S, ET => TimerON_0); // TON
R_TRIG_7(CLK := TON_0.Q AND SOP640_B6); // R_TRIG
_w4 := R_TRIG_7.Q;
IF _w4 THEN SOP640_pmsg := 'WARNING: PRODUCTION STOPPED - BOX WAITING'; END_IF
SOP640_RS S= _w4;
SOP640_BoxWaiting S= _w4;
R_TRIG_8(CLK := TON_0.Q AND NOT SOP640_B6); // R_TRIG
_w5 := R_TRIG_8.Q;
IF _w5 THEN SOP640_pmsg := 'ALARM: PRODUCTION STOPPED - BOX WAITING'; END_IF
SOP640_RS S= _w5;
SOP640_BoxWaiting S= _w5;
_w6 := NOT SOP640_Occupied AND SOP640_BoxWaiting;
IF _w6 THEN SOP640_pmsg := 'No Alarms'; END_IF
SOP640_RS S= _w6;
SOP640_BoxWaiting R= _w6;

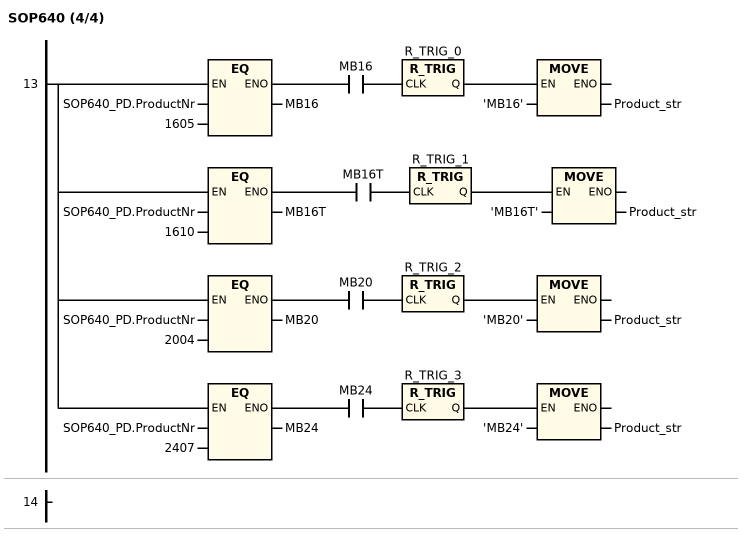
// NETWORK 13
MB16 := SOP640_PD.ProductNr = 1605;
R_TRIG_0(CLK := MB16); // R_TRIG
_w7 := R_TRIG_0.Q;
IF _w7 THEN Product_str := 'MB16'; END_IF
MB16T := SOP640_PD.ProductNr = 1610;
R_TRIG_1(CLK := MB16T); // R_TRIG
_w8 := R_TRIG_1.Q;
IF _w8 THEN Product_str := 'MB16T'; END_IF
MB20 := SOP640_PD.ProductNr = 2004;
R_TRIG_2(CLK := MB20); // R_TRIG
_w9 := R_TRIG_2.Q;
IF _w9 THEN Product_str := 'MB20'; END_IF
MB24 := SOP640_PD.ProductNr = 2407;
R_TRIG_3(CLK := MB24); // R_TRIG
_w10 := R_TRIG_3.Q;
IF _w10 THEN Product_str := 'MB24'; END_IF
(* _w7 OR _w8 OR _w9 OR _w10; result not used *)

// NETWORK 14

END_PROGRAM

// Device/Application/FBs/FB_InspectionConveyor
FUNCTION_BLOCK FB_InspectionConveyor
VAR_INPUT
	iAuto_On: BOOL; // Auto-On cycle active
	iHoming_On: BOOL; // Homing-On cycle active
	iManual: BOOL; // Manual mode active
	iSafety_OK: BOOL; // Safety circuit OK
	iStop_EOC: BOOL; // Stop EOC selected
	iResetAlarms: BOOL; // Reset Alarms
	
	iEnFwd: BOOL := TRUE; // Interlock signal movement forward
	iEnRev: BOOL := TRUE; // Interlock signal movement reverse
	
	iMFwd: BOOL; 	// Manual Fwd request
	iMRev: BOOL; 	// Manual Rev request
	iMFrontClampUp: BOOL; 	// Manual Front Clamp Up request
	iMFrontClampDown: BOOL; 	// Manual Front Clamp Down request
	iMRearClampUp: BOOL; 	// Manual Front Clamp Up request
	iMRearClampDown: BOOL; 	// Manual Front Clamp Down request
	iMPDFwd: BOOL; 	// Manual Move PD forward
	iMPDRev: BOOL; 	// Manual Move PD reverse
	
	iProtectionTripped: BOOL := FALSE; // Motor Protection Tripped
	
	iSensorPos: BOOL; // Product in position
	iFrontClampDown: BOOL; // Front Clamp in lower position
	iFrontClampUp: BOOL; // Front Clamp in upper position
	iRearClampDown: BOOL; // Rear Clamp in lower position
	iRearClampUp: BOOL; // Rear Clamp in upper position
	
	iEnTravelIn: BOOL := TRUE; // Enable product transfer from previous conveyor.
	iEnTravelOut: BOOL := TRUE; // Enable product transfer to next conveyor.
	
	iPrevReadyToTransfer: BOOL; // Previous conveyor ready to transfer
	iPrevTransfering: BOOL; // Previous conveyor transfering
	iNextTransferOK: BOOL; // Next conveyor ready to load
	iNextTransferDone: BOOL;  // Next conveyor transfer done
	
	iTimeOutTransferIn: TIME := T#10S; // Time out time for transfer in
	iTimeOutTransferOut: TIME := T#10S; // Time out time for transfer out
	iTimeOutFrontClamp: TIME := T#3S; // Time out time for Front Clamp Cylinder
	iTimeOutRearClamp: TIME := T#3S; // Time out time for Rear Clamp Cylinder
END_VAR
VAR_IN_OUT
	ProductionData: ProductionData; 		// Production Data
	Prev_ProductionData: ProductionData;	// Previous Production Data
	Next_ProductionData: ProductionData;	// Next Production Data
END_VAR
VAR_OUTPUT
	oRunning: BOOL; // Conveyor Running
	oOccupied: BOOL; // Conveyor Occupied
	oFaulted : BOOL; // Conveyor faulted
	oFault_Code: INT; // Conveyor fault code
	oHome_Pos: BOOL; // Conveyor Home Position reached
	oEOC_Pos: BOOL; // Conveyor Stop EOC reached

	oRunFwd: BOOL; // Conveyor running forward
	oRunRev: BOOL; // Conveyor running reverse	

	oFrontClampUp: BOOL; // Front Clamping Cylinder Up
	oFrontClampDown: BOOL; // Front Clamping Cylinder Down	
	oRearClampUp: BOOL; // Rear Clamping Cylinder Up
	oRearClampDown: BOOL; // Rear Clamping Cylinder Down	

	oPrevTransferOK: BOOL; // Conveyor ready to load
	oPrevTransferDone: BOOL; // Conveyor load completed
	oNextReadyToTransfer: BOOL; // Conveyor ready to transfer
	oNextTransfering: BOOL; // Conveyor transfering
END_VAR
VAR
	AutoSteps: WORD;
	HomeSteps: WORD;
	
	Timeout_Fault1: TON;
	Timeout_Fault2: TON;
	
	EmptyPD: ProductionData;
	PDValid: BOOL;		// PD is Valid
	PDEmpty: BOOL;		// PD is Empty
	PrevPDValid: BOOL;	// Previous PD is Valid
	PrevPDEmpty: BOOL;	// Previous PD is Empty
	NextPDValid: BOOL;	// Next PD is Valid
	NextPDEmpty: BOOL;	// Next PD is Empty
	R_TRIG_TransferPDFwd: R_TRIG;
	R_TRIG_TransferPDRev: R_TRIG;
	R_TRIG_Fault_10: R_TRIG;
	R_TRIG_Fault_11: R_TRIG;
	R_TRIG_Fault_12: R_TRIG;
	iMFrontClampFwd: BOOL;
	Timeout_Fault3: TON;
	Timeout_Fault4: TON;
END_VAR
VAR // added by the converter: edge detectors and wires of the graphical bodies
    _w1, _w2, _w3, _w4, _w5, _w6, _w7, _w8, _w9, _w10, _w11, _w12, _w13, _w14, _w15, _w16, _w17, _w18, _w19, _w20, _w21 : BOOL;
END_VAR

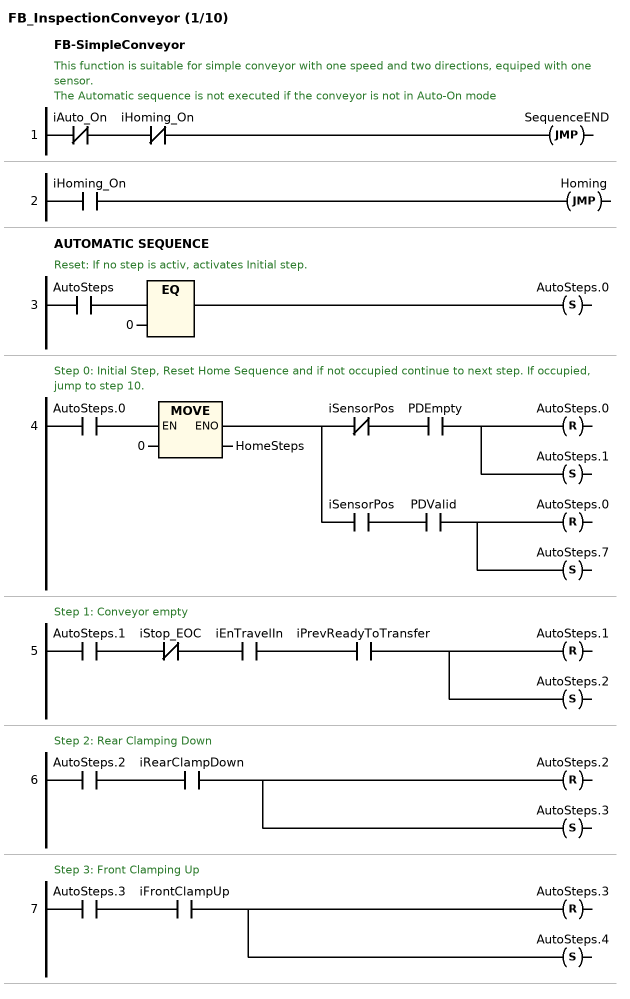
// NETWORK 1: FB-SimpleConveyor
// This function is suitable for simple conveyor with one speed and two directions, equiped with one sensor.
//
// The Automatic sequence is not executed if the conveyor is not in Auto-On mode
IF NOT iAuto_On AND NOT iHoming_On THEN JMP SequenceEND; END_IF

// NETWORK 2
IF iHoming_On THEN JMP Homing; END_IF

// NETWORK 3: AUTOMATIC SEQUENCE
// Reset: If no step is activ, activates Initial step.
AutoSteps.0 S= AutoSteps = 0;

// NETWORK 4
// Step 0: Initial Step, Reset Home Sequence and if not occupied continue to next step. If occupied, jump to step 10.
_w1 := AutoSteps.0;
IF _w1 THEN HomeSteps := 0; END_IF
_w2 := _w1 AND NOT iSensorPos AND PDEmpty;
AutoSteps.0 R= _w2;
AutoSteps.1 S= _w2;
_w3 := _w1 AND iSensorPos AND PDValid;
AutoSteps.0 R= _w3;
AutoSteps.7 S= _w3;

// NETWORK 5
// Step 1: Conveyor empty
_w4 := AutoSteps.1 AND NOT iStop_EOC AND iEnTravelIn AND iPrevReadyToTransfer;
AutoSteps.1 R= _w4;
AutoSteps.2 S= _w4;

// NETWORK 6
// Step 2: Rear Clamping Down
_w5 := AutoSteps.2 AND iRearClampDown;
AutoSteps.2 R= _w5;
AutoSteps.3 S= _w5;

// NETWORK 7
// Step 3: Front Clamping Up
_w6 := AutoSteps.3 AND iFrontClampUp;
AutoSteps.3 R= _w6;
AutoSteps.4 S= _w6;

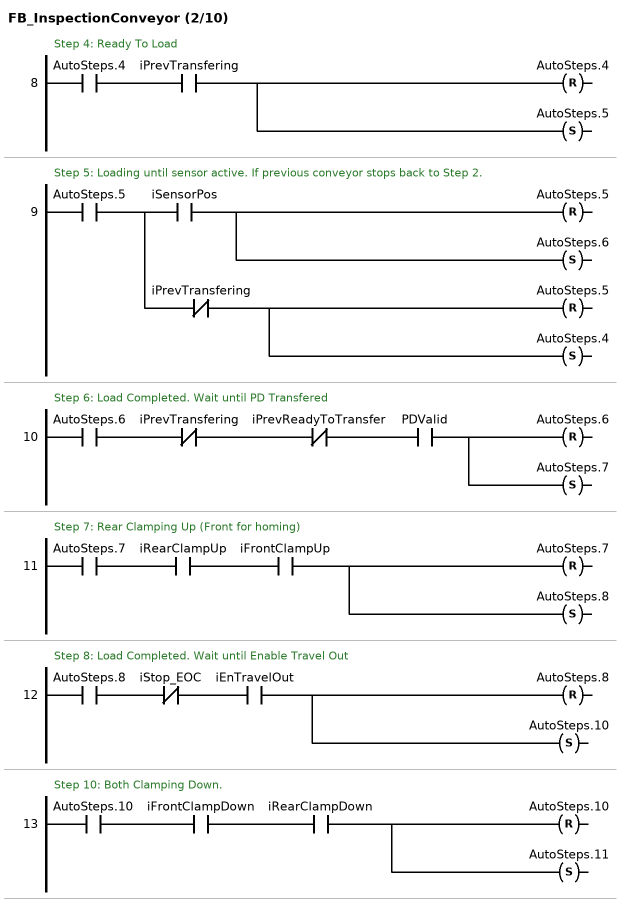
// NETWORK 8
// Step 4: Ready To Load
_w7 := AutoSteps.4 AND iPrevTransfering;
AutoSteps.4 R= _w7;
AutoSteps.5 S= _w7;

// NETWORK 9
// Step 5: Loading until sensor active. If previous conveyor stops back to Step 2.
_w8 := AutoSteps.5;
_w9 := _w8 AND iSensorPos;
AutoSteps.5 R= _w9;
AutoSteps.6 S= _w9;
_w10 := _w8 AND NOT iPrevTransfering;
AutoSteps.5 R= _w10;
AutoSteps.4 S= _w10;

// NETWORK 10
// Step 6: Load Completed. Wait until PD Transfered
_w11 := AutoSteps.6 AND NOT iPrevTransfering AND NOT iPrevReadyToTransfer AND PDValid;
AutoSteps.6 R= _w11;
AutoSteps.7 S= _w11;

// NETWORK 11
// Step 7: Rear Clamping Up (Front for homing)
_w12 := AutoSteps.7 AND iRearClampUp AND iFrontClampUp;
AutoSteps.7 R= _w12;
AutoSteps.8 S= _w12;

// NETWORK 12
// Step 8: Load Completed. Wait until Enable Travel Out
_w13 := AutoSteps.8 AND NOT iStop_EOC AND iEnTravelOut;
AutoSteps.8 R= _w13;
AutoSteps.10 S= _w13;

// NETWORK 13
// Step 10: Both Clamping Down.
_w14 := AutoSteps.10 AND iFrontClampDown AND iRearClampDown;
AutoSteps.10 R= _w14;
AutoSteps.11 S= _w14;

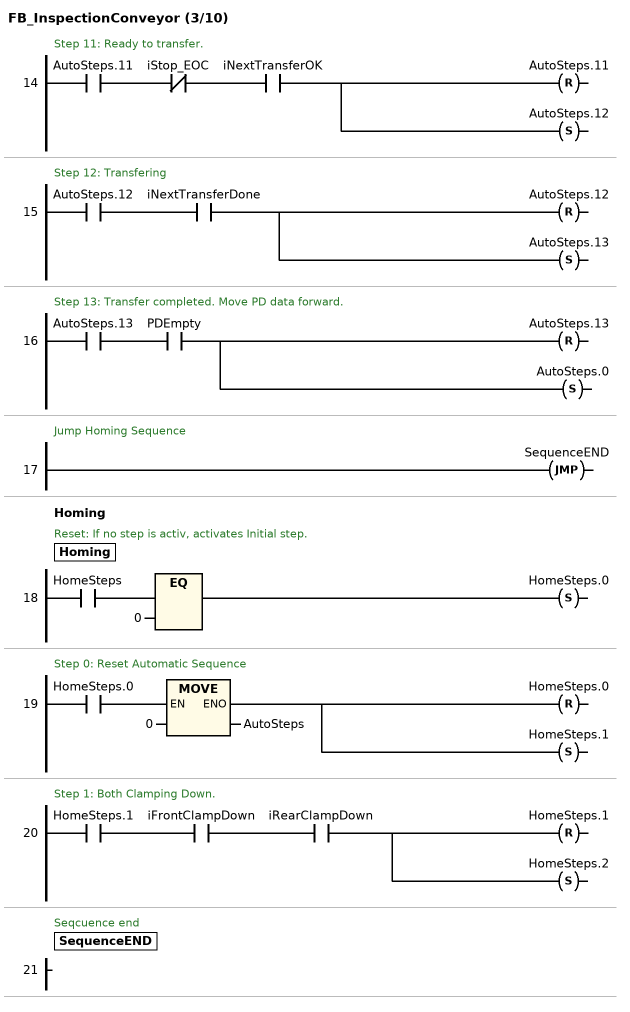
// NETWORK 14
// Step 11: Ready to transfer.
_w15 := AutoSteps.11 AND NOT iStop_EOC AND iNextTransferOK;
AutoSteps.11 R= _w15;
AutoSteps.12 S= _w15;

// NETWORK 15
// Step 12: Transfering
_w16 := AutoSteps.12 AND iNextTransferDone;
AutoSteps.12 R= _w16;
AutoSteps.13 S= _w16;

// NETWORK 16
// Step 13: Transfer completed. Move PD data forward.
_w17 := AutoSteps.13 AND PDEmpty;
AutoSteps.13 R= _w17;
AutoSteps.0 S= _w17;

// NETWORK 17
// Jump Homing Sequence
JMP SequenceEND;

// NETWORK 18: Homing
// Reset: If no step is activ, activates Initial step.
Homing:
HomeSteps.0 S= HomeSteps = 0;

// NETWORK 19
// Step 0: Reset Automatic Sequence
_w18 := HomeSteps.0;
IF _w18 THEN AutoSteps := 0; END_IF
HomeSteps.0 R= _w18;
HomeSteps.1 S= _w18;

// NETWORK 20
// Step 1: Both Clamping Down.
_w19 := HomeSteps.1 AND iFrontClampDown AND iRearClampDown;
HomeSteps.1 R= _w19;
HomeSteps.2 S= _w19;

// NETWORK 21
// Seqcuence end
SequenceEND: ;

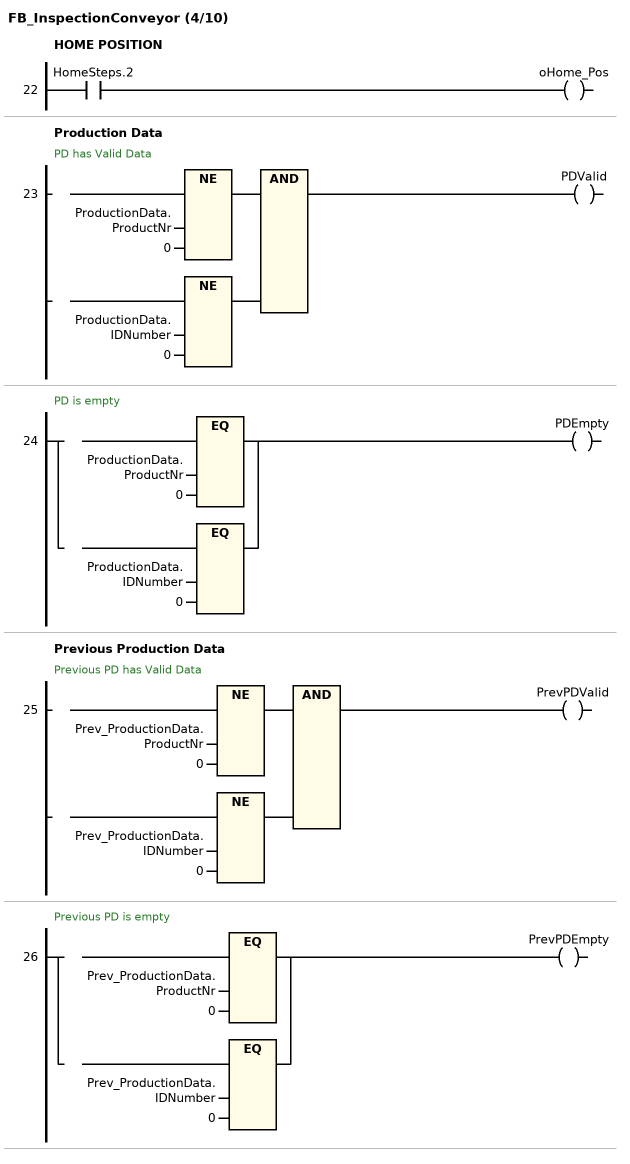
// NETWORK 22: HOME POSITION
oHome_Pos := HomeSteps.2;

// NETWORK 23: Production Data
// PD has Valid Data
PDValid := ProductionData.ProductNr <> 0 AND ProductionData.IDNumber <> 0;

// NETWORK 24
// PD is empty
PDEmpty := ProductionData.ProductNr = 0 OR ProductionData.IDNumber = 0;

// NETWORK 25: Previous Production Data
// Previous PD has Valid Data
PrevPDValid := Prev_ProductionData.ProductNr <> 0 AND Prev_ProductionData.IDNumber <> 0;

// NETWORK 26
// Previous PD is empty
PrevPDEmpty := Prev_ProductionData.ProductNr = 0 OR Prev_ProductionData.IDNumber = 0;

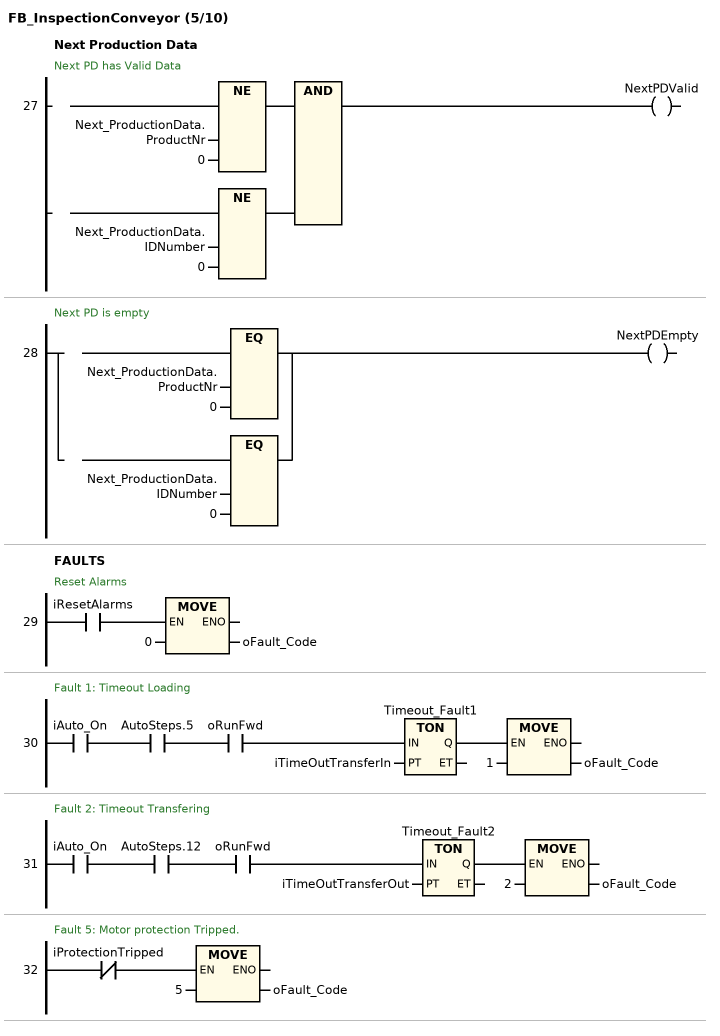
// NETWORK 27: Next Production Data
// Next PD has Valid Data
NextPDValid := Next_ProductionData.ProductNr <> 0 AND Next_ProductionData.IDNumber <> 0;

// NETWORK 28
// Next PD is empty
NextPDEmpty := Next_ProductionData.ProductNr = 0 OR Next_ProductionData.IDNumber = 0;

// NETWORK 29: FAULTS
// Reset Alarms
IF iResetAlarms THEN oFault_Code := 0; END_IF

// NETWORK 30
// Fault 1: Timeout Loading
Timeout_Fault1(IN := iAuto_On AND AutoSteps.5 AND oRunFwd, PT := iTimeOutTransferIn); // TON
IF Timeout_Fault1.Q THEN oFault_Code := 1; END_IF

// NETWORK 31
// Fault 2: Timeout Transfering
Timeout_Fault2(IN := iAuto_On AND AutoSteps.12 AND oRunFwd, PT := iTimeOutTransferOut); // TON
IF Timeout_Fault2.Q THEN oFault_Code := 2; END_IF

// NETWORK 32
// Fault 5: Motor protection Tripped.
IF NOT iProtectionTripped THEN oFault_Code := 5; END_IF

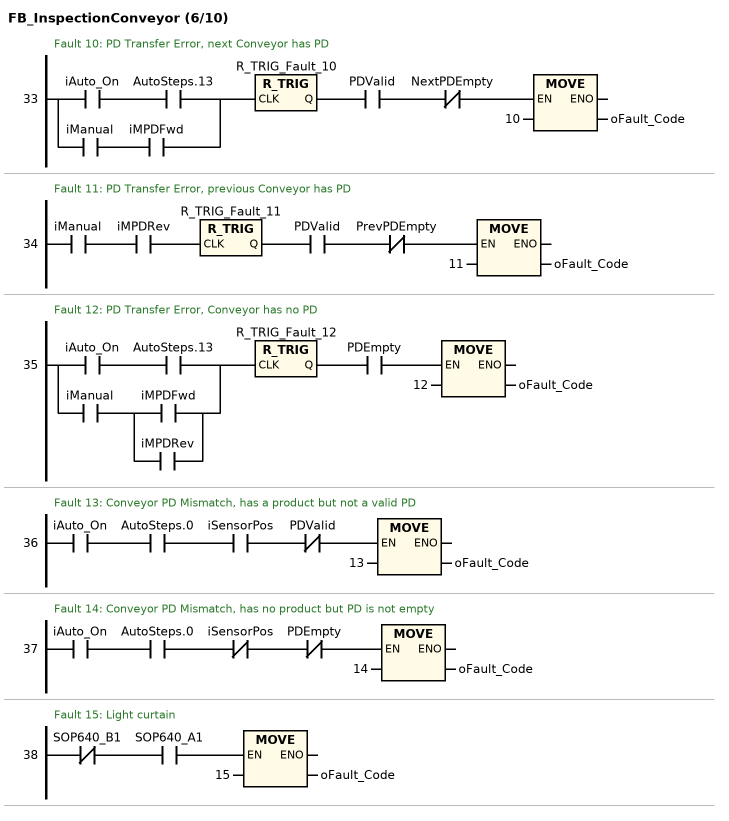
// NETWORK 33
// Fault 10: PD Transfer Error, next Conveyor has PD
R_TRIG_Fault_10(CLK := iAuto_On AND AutoSteps.13 OR iManual AND iMPDFwd); // R_TRIG
IF R_TRIG_Fault_10.Q AND PDValid AND NOT NextPDEmpty THEN oFault_Code := 10; END_IF

// NETWORK 34
// Fault 11: PD Transfer Error, previous Conveyor has PD
R_TRIG_Fault_11(CLK := iManual AND iMPDRev); // R_TRIG
IF R_TRIG_Fault_11.Q AND PDValid AND NOT PrevPDEmpty THEN oFault_Code := 11; END_IF

// NETWORK 35
// Fault 12: PD Transfer Error, Conveyor has no PD
R_TRIG_Fault_12(CLK := iAuto_On AND AutoSteps.13 OR iManual AND (iMPDFwd OR iMPDRev)); // R_TRIG
IF R_TRIG_Fault_12.Q AND PDEmpty THEN oFault_Code := 12; END_IF

// NETWORK 36
// Fault 13: Conveyor PD Mismatch, has a product but not a valid PD
IF iAuto_On AND AutoSteps.0 AND iSensorPos AND NOT PDValid THEN oFault_Code := 13; END_IF

// NETWORK 37
// Fault 14: Conveyor PD Mismatch, has no product but PD is not empty
IF iAuto_On AND AutoSteps.0 AND NOT iSensorPos AND NOT PDEmpty THEN oFault_Code := 14; END_IF

// NETWORK 38
// Fault 15: Light curtain
IF NOT SOP640_B1 AND SOP640_A1 THEN oFault_Code := 15; END_IF

